FUNCTION_BLOCK Wrapper
VAR_INPUT
	ActInputs   : ActInputs;
	Buttons		: Buttons;  
END_VAR
VAR_OUTPUT
	ActOutputs	: ActOutputs;
	Flags		: Flags;
END_VAR
VAR	
	ButtonCheck		: ButtonCheck;

	Gripper			: Gripper;
	HorizontalAct	: HorizontalAct;
	VerticalAct		: VerticalAct;
	CellSensor		: CellSensor;
	CycleCount		: CycleCount;
END_VAR

METHOD mMap : BOOL
VAR_INPUT
END_VAR
/////// Inputs //////////
Gripper.pClosed		:= ActInputs.Closed;
Gripper.pOpened		:= ActInputs.Opened;
HorizontalAct.pExtended		:= ActInputs.Extended;
HorizontalAct.pRetracted	:= ActInputs.Retracted;
VerticalAct.pLowered	:= ActInputs.Lowered;
VerticalAct.pRaised		:= ActInputs.Raised;
ButtonCheck.pEStop	:= Buttons.EStop;
ButtonCheck.pReset	:= Buttons.Reset;
ButtonCheck.pStart	:= Buttons.Start;

/////// Outputs //////////
ActOutputs.Close 	:= Gripper.pClose;
ActOutputs.Extend	:= HorizontalAct.pExtend;
ActOutputs.Raise	:= VerticalAct.pRaise;
Flags.PartReady 	:= CellSensor.pFeeded;
Flags.PlaceReady	:= CellSensor.pOKtoRelase;
Flags.Picked		:= CycleCount.pPicked;
END_METHOD

END_FUNCTION_BLOCK

(* stored: Version 1.1.0.1, ProductVersion 3.1.4024.9
   POU Wrapper: Id {0bc2863a-f0e7-4344-aff6-4cc0fac2d441}, SpecialFunc None
   Method mMap: Id {660594b9-b959-4881-8851-34fbe3841409} *)
